Staubli VAL3: actBtnFinished.pgx

program actBtnFinished()
begin
  bFinished=true
end
